(*
	
*)

FUNCTION_BLOCK RecordDataQueue IMPLEMENTS IRecordDataQueue
VAR
	current_index	: UDINT; // current index value
	sMeasurementName			: Tc2_System.T_MaxString;	// Measurement name of InfluxDB
	sSchemaName					: Tc2_System.T_MaxString;	// Schema name as a inserted data variable type name as structure
	min_chunk_size				: UDINT := 300;				// Minimum chunk size
	max_chunk_size				:UDINT	:= 10000;			// Maximum chunk size
	nDataBufferMaxIndex			: UDINT := 1;				// upper bound of data buffer array.			
	gRecordPointer				: Tc2_Utilities.T_Arg;		// Current data index
	// Variables for queue feature
	get_data_t 		: T_Arg;
	get_data 		: DbInsertCommand;
	
	// Start point time
	start_time		: ULINT;
	start_data 		: T_Arg;

	nCycleTime		: UDINT;					// PLC task cycle time setting(in 100ns)
	data_size		: UDINT := 1;				// record data size
	data_count		: UDINT := 0;		// buffer usage
	last_data_count	: UDINT := 0;
	
	start_index		: UDINT;
	_buffer_usage	: REAL;				// data usage percentage of data buffer.
	_avalable_buffer_size	:DINT;
	diff_target		: REAL;
	pid_ope			: REAL;	
	recording		: BOOL;
	chunk_size : UDINT;
	bContinue		: BOOL;
	//insert_command_buffer	: ARRAY [0..QUEUE_SIZE] OF DbInsertCommand;
	//BufferIndex			: ARRAY [0..QUEUE_SIZE] OF T_Arg;
	insert_command_buffer: INT;
	
END_VAR

VAR_OUTPUT
	next_index 		: UDINT;
END_VAR

VAR_IN_OUT
	command_queue 	: CommandQueueMember;	// Queue members for shared.
END_VAR

PROPERTY PUBLIC buffer_usage : REAL
GET
buffer_usage := _buffer_usage;
END_GET
SET
END_SET
END_PROPERTY

// Explicity specify cycle time.
PROPERTY PUBLIC cycle_time : UDINT
GET
END_GET
SET
nCycleTime := cycle_time;
END_SET
END_PROPERTY

METHOD cyclic_record : BOOL
VAR_INPUT
END_VAR
IF current_index = start_index THEN
	start_time := F_GetSystemTime();
	start_data := gRecordPointer;
END_IF

IF next_index <= current_index OR current_index >= nDataBufferMaxIndex THEN
	max_chunk_size := nDataBufferMaxIndex + 1;
	// put_data
	IF NOT command_queue.controller.full THEN
		data_size := current_index - start_index + 1;
		_avalable_buffer_size := UDINT_TO_DINT(nDataBufferMaxIndex) - UDINT_TO_DINT(data_count) +1;
		IF _avalable_buffer_size < UDINT_TO_DINT(data_size) AND _avalable_buffer_size > 0 THEN
			data_size := DINT_TO_UDINT(_avalable_buffer_size);
		ELSIF _avalable_buffer_size <= 0 THEN
			data_size := 0;
		END_IF

		IF data_size > 1 THEN

			// put pointer
			IF command_queue.current_index > command_queue.buffer_size THEN
				command_queue.current_index := 0;
			END_IF
			
			// calculate each cycle time by num of data among start time and current time.
			nCycleTime := ULINT_TO_UDINT(F_GetSystemTime() - start_time) / (data_size - 1);
		
			// set value of insert command
			command_queue.buffer_body[command_queue.current_index].data_body := start_data;
			command_queue.buffer_body[command_queue.current_index].start_time := start_time;
			command_queue.buffer_body[command_queue.current_index].cycle_time_100ns := nCycleTime;
			command_queue.buffer_body[command_queue.current_index].chunk_size := data_size;
			command_queue.buffer_body[command_queue.current_index].MeasurementName := sMeasurementName;
			command_queue.buffer_body[command_queue.current_index].SchemaName := sSchemaName;
			command_queue.buffer_body[command_queue.current_index].ref_data_buffer_counter REF= data_count;
			// queue in
			command_queue.controller.put(
				lData := F_BIGTYPE(
					pData := ADR(command_queue.buffer_body[command_queue.current_index]), 
					cbLen := SIZEOF(command_queue.buffer_body[command_queue.current_index])
				)
			);
			data_count := data_count + command_queue.buffer_body[command_queue.current_index].chunk_size;
			command_queue.current_index := command_queue.current_index + 1;
			start_index := current_index + 1;
		END_IF
	END_IF
END_IF


IF last_data_count <> data_count THEN
	// calculate next index
	_buffer_usage := UDINT_TO_REAL(data_count) / UDINT_TO_REAL(nDataBufferMaxIndex + 1);
	diff_target := UDINT_TO_REAL(max_chunk_size) * _buffer_usage;
	pid_ope := UDINT_TO_REAL(min_chunk_size) + diff_target;
	chunk_size := REAL_TO_UDINT(pid_ope);
	//chunk_size := minimum_chunk_size;
	next_index := current_index + chunk_size - 1;
	IF chunk_size < min_chunk_size OR pid_ope < 0 THEN
		chunk_size := min_chunk_size;
	ELSIF chunk_size > max_chunk_size THEN
		chunk_size := max_chunk_size;
	END_IF
END_IF

last_data_count := data_count;

IF current_index < nDataBufferMaxIndex THEN
	current_index := current_index + 1;
ELSE
	current_index := 0;
	start_index := 0;
	next_index := chunk_size - 1;
END_IF
END_METHOD

PROPERTY PUBLIC data_def_structure_name : Tc2_System.T_MaxString
GET
END_GET
SET
sSchemaName := data_def_structure_name;
END_SET
END_PROPERTY

PROPERTY PUBLIC data_pointer : T_Arg
GET
data_pointer := gRecordPointer;
END_GET
SET
gRecordPointer := data_pointer;
END_SET
END_PROPERTY

PROPERTY PUBLIC db_table_name : Tc2_System.T_MaxString
GET
END_GET
SET
sMeasurementName := db_table_name;
END_SET
END_PROPERTY

PROPERTY PUBLIC index : UDINT
GET
index := current_index;
END_GET
SET
END_SET
END_PROPERTY

PROPERTY PUBLIC maximum_chunk_size : UDINT
GET
maximum_chunk_size := max_chunk_size;
END_GET
SET
max_chunk_size := maximum_chunk_size;
END_SET
END_PROPERTY

PROPERTY PUBLIC minimum_chunk_size : UDINT
GET
minimum_chunk_size := min_chunk_size;
END_GET
SET
min_chunk_size := minimum_chunk_size;
END_SET
END_PROPERTY

(*
Command will be generated once.

Data insert command will be generated at every cycle. 

*)

METHOD record_once : BOOL
VAR_INPUT
END_VAR
// put_data
IF NOT command_queue.controller.full THEN
	// put pointer
	IF command_queue.current_index > command_queue.buffer_size THEN
		command_queue.current_index := 0;
	END_IF
	
	// set value of insert command
	command_queue.buffer_body[command_queue.current_index].data_body := gRecordPointer;
	command_queue.buffer_body[command_queue.current_index].start_time := F_GetSystemTime();
	command_queue.buffer_body[command_queue.current_index].cycle_time_100ns := nCycleTime;
	command_queue.buffer_body[command_queue.current_index].chunk_size := data_size;
	command_queue.buffer_body[command_queue.current_index].MeasurementName := sMeasurementName;
	command_queue.buffer_body[command_queue.current_index].SchemaName := sSchemaName;
	command_queue.buffer_body[command_queue.current_index].ref_data_buffer_counter REF= data_count;
	// queue in
	IF  data_size <= (nDataBufferMaxIndex - data_count) THEN
		command_queue.controller.put(
			lData := F_BIGTYPE(
				pData := ADR(command_queue.buffer_body[command_queue.current_index]), 
				cbLen := SIZEOF(command_queue.buffer_body[command_queue.current_index])
			)
		);
		data_count := data_count + command_queue.buffer_body[command_queue.current_index].chunk_size;
		command_queue.current_index := command_queue.current_index + 1;
	END_IF
END_IF
END_METHOD

PROPERTY PUBLIC upper_bound_of_data_buffer : UDINT
GET
END_GET
SET
nDataBufferMaxIndex := upper_bound_of_data_buffer;
END_SET
END_PROPERTY

END_FUNCTION_BLOCK

(* stored: Version 1.1.0.1, ProductVersion 3.1.4024.12
   POU RecordDataQueue: Id {8b3999e3-c2e1-4344-9092-4e707723d89a}, SpecialFunc None
   Property buffer_usage: Id {bbb95211-74e1-4da1-9e2b-be2248fb01e5}
   Get Get: Id {b46d5d51-f7df-45ba-9aab-0d3c72cb9324}
   Set Set: Id {c88e0f39-ef98-4aac-999b-7b9e79aeaac6}
   Property cycle_time: Id {dd6efd39-1e93-4941-82d8-5c6febd1514f}
   Get Get: Id {544d71c5-8eb0-4fef-a4dc-9a6773175e9a}
   Set Set: Id {5587682c-4f41-4fa1-bbe3-a995cd57dc9a}
   Method cyclic_record: Id {4d6a4f57-2187-4032-b3a4-3e31e3263b61}
   Property data_def_structure_name: Id {12d15a2c-bf0d-4db7-a907-7cebd338c4d6}
   Get Get: Id {ebda072e-3d15-41ca-8ab8-cbbe755d7e35}
   Set Set: Id {374779eb-84af-449b-b1d1-d49d94a7b136}
   Property data_pointer: Id {07abae9f-fcfc-4930-be5e-bc498c167473}
   Get Get: Id {91fd2a72-f38a-48ad-a8d9-3b379b6c1197}
   Set Set: Id {4c0a6bcb-e79a-4e5a-a3b2-b65082e77189}
   Property db_table_name: Id {457088bd-30e0-4a96-b934-15df6743d6b6}
   Get Get: Id {4d8d5759-a539-49cb-92e4-0c653a06c4e1}
   Set Set: Id {5583acd3-dff8-4ba3-acf1-2446e6b0a828}
   Property index: Id {2cd967fd-5fa9-4645-9ac7-7c80e69c201d}
   Get Get: Id {0b55b3f6-4958-4ca5-9778-68f6ede6f192}
   Set Set: Id {5268f547-a543-47a9-b5ad-fb8f56729f3a}
   Property maximum_chunk_size: Id {02c2c686-c7db-499b-a50c-3e861736b577}
   Get Get: Id {0baff072-67eb-4a7c-8fad-76d523574483}
   Set Set: Id {59369926-4939-4df1-910f-88ccb0b731a6}
   Property minimum_chunk_size: Id {7194ace4-c543-4d3b-bb4c-7732e82ecf0f}
   Get Get: Id {a7346a3e-d6df-4d67-acd9-15108b0b7d1f}
   Set Set: Id {bf381183-3550-45b7-9d0d-d87b431cae4d}
   Method record_once: Id {de86fac9-c1d3-47d8-8df5-68c1cbb5521d}
   Property upper_bound_of_data_buffer: Id {f8195cd1-4b1c-4c66-b057-b390adf2edea}
   Get Get: Id {3661889e-c6c5-41e5-ac1c-840bad373726}
   Set Set: Id {90946641-4400-49dd-b911-8d0d9ebdf329} *)
